PROGRAM ladder_logic_diagram 
VAR
	t2s: TIME := TIME#3S;
	t0s: TIME := TIME#0S;
	Timer: TON;
	input : BOOL;
	output : BOOL; 
	TON_Reset: TON;
	TON_set: TON;
	TON_0: TON;
	TON_Trig: TON;
	TON_Autonomous: TON;
	TON_Manual: TON;
	TON_Lock: TON;
	Robot_Mode_Timer: TON;
	liftUP: TON;
	liftDOWN: TON;
	load_button  AT %I* : BOOL ;
	load_active AT %Q*: BOOL;
	trigger AT %M* : BOOL ;
	T: TIME;
	TON_1: TON;
	TON2: TON;
	TON_3: TON;
	activate_time_read: BOOL;
	TON_4: TON;
	second_read_triggered: BOOL;
	first_read_triggered: BOOL;
	TON_5: TON;
	TON_6: TON;
	TON_7: TON;
END_VAR
VAR // added by the converter: edge detectors and wires of the graphical bodies
    _rt1 : R_TRIG;
    _w1 : BOOL;
END_VAR

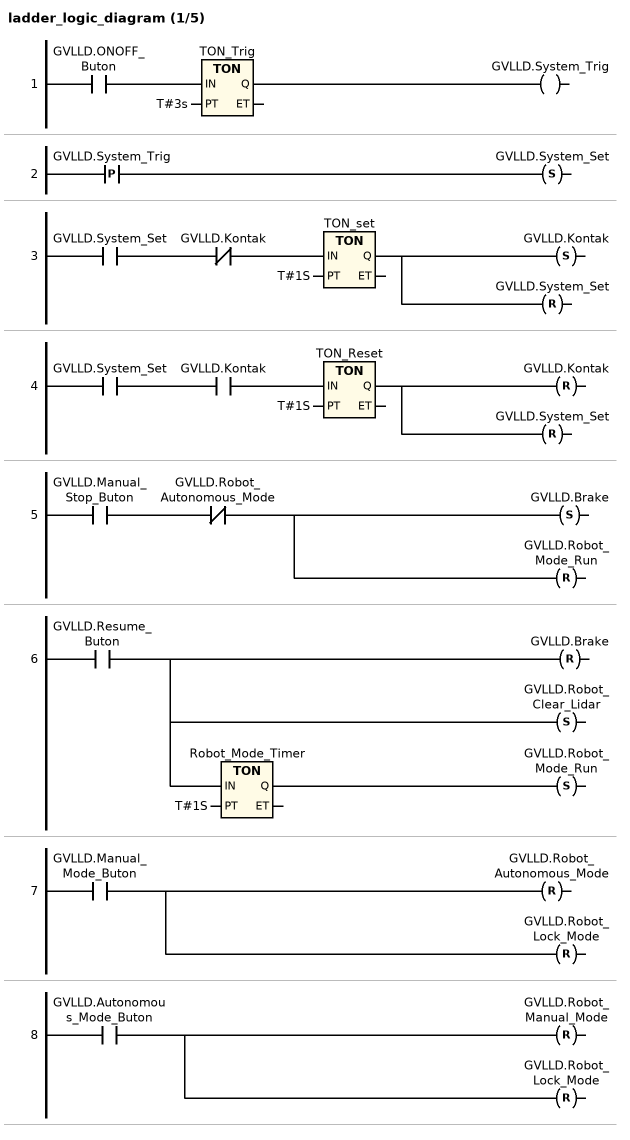
// NETWORK 1
TON_Trig(IN := GVLLD.ONOFF_Buton, PT := T#3s); // TON
GVLLD.System_Trig := TON_Trig.Q;

// NETWORK 2
_rt1(CLK := GVLLD.System_Trig);
GVLLD.System_Set S= _rt1.Q;

// NETWORK 3
TON_set(IN := GVLLD.System_Set AND NOT GVLLD.Kontak, PT := T#1S); // TON
GVLLD.Kontak S= TON_set.Q;
GVLLD.System_Set R= TON_set.Q;

// NETWORK 4
TON_Reset(IN := GVLLD.System_Set AND GVLLD.Kontak, PT := T#1S); // TON
GVLLD.Kontak R= TON_Reset.Q;
GVLLD.System_Set R= TON_Reset.Q;

// NETWORK 5
_w1 := GVLLD.Manual_Stop_Buton AND NOT GVLLD.Robot_Autonomous_Mode;
GVLLD.Brake S= _w1;
GVLLD.Robot_Mode_Run R= _w1;

// NETWORK 6
GVLLD.Brake R= GVLLD.Resume_Buton;
GVLLD.Robot_Clear_Lidar S= GVLLD.Resume_Buton;
Robot_Mode_Timer(IN := GVLLD.Resume_Buton, PT := T#1S); // TON
GVLLD.Robot_Mode_Run S= Robot_Mode_Timer.Q;

// NETWORK 7
GVLLD.Robot_Autonomous_Mode R= GVLLD.Manual_Mode_Buton;
GVLLD.Robot_Lock_Mode R= GVLLD.Manual_Mode_Buton;

// NETWORK 8
GVLLD.Robot_Manual_Mode R= GVLLD.Autonomous_Mode_Buton;
GVLLD.Robot_Lock_Mode R= GVLLD.Autonomous_Mode_Buton;

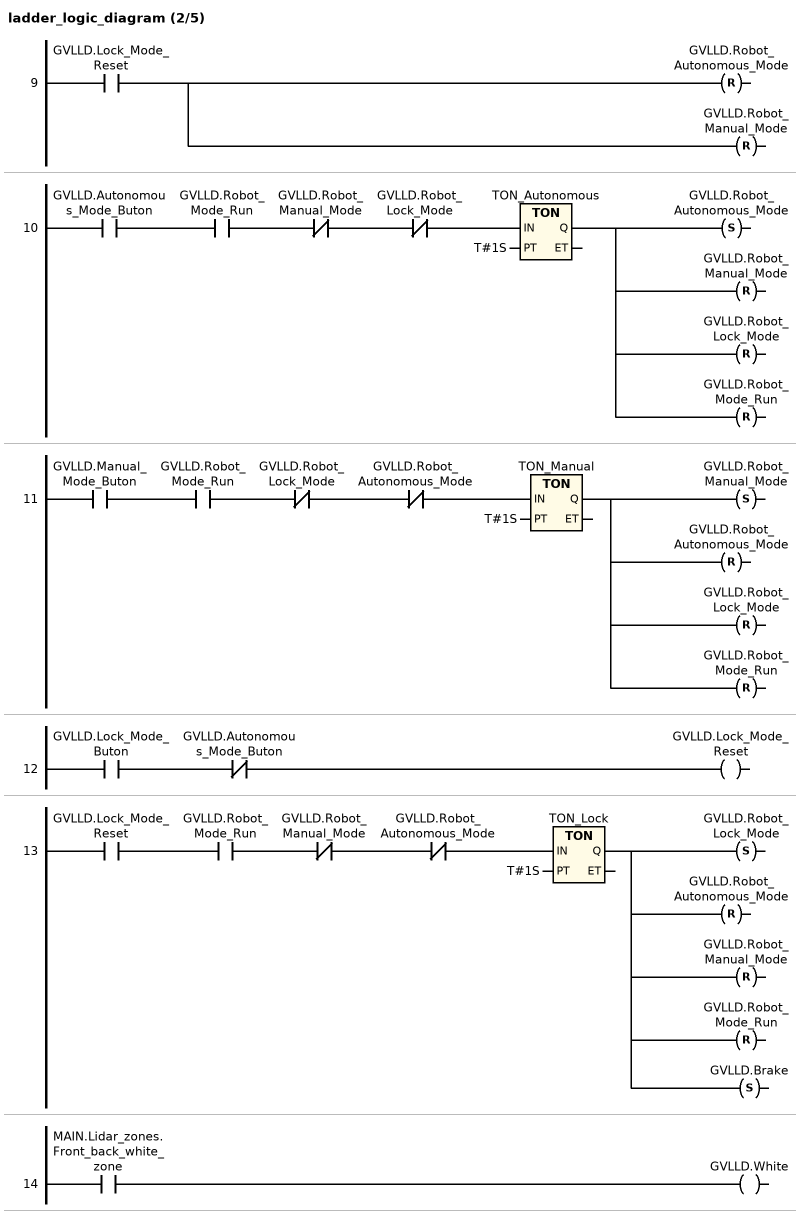
// NETWORK 9
GVLLD.Robot_Autonomous_Mode R= GVLLD.Lock_Mode_Reset;
GVLLD.Robot_Manual_Mode R= GVLLD.Lock_Mode_Reset;

// NETWORK 10
TON_Autonomous(IN := GVLLD.Autonomous_Mode_Buton AND GVLLD.Robot_Mode_Run AND NOT GVLLD.Robot_Manual_Mode AND NOT GVLLD.Robot_Lock_Mode, PT := T#1S); // TON
GVLLD.Robot_Autonomous_Mode S= TON_Autonomous.Q;
GVLLD.Robot_Manual_Mode R= TON_Autonomous.Q;
GVLLD.Robot_Lock_Mode R= TON_Autonomous.Q;
GVLLD.Robot_Mode_Run R= TON_Autonomous.Q;

// NETWORK 11
TON_Manual(IN := GVLLD.Manual_Mode_Buton AND GVLLD.Robot_Mode_Run AND NOT GVLLD.Robot_Lock_Mode AND NOT GVLLD.Robot_Autonomous_Mode, PT := T#1S); // TON
GVLLD.Robot_Manual_Mode S= TON_Manual.Q;
GVLLD.Robot_Autonomous_Mode R= TON_Manual.Q;
GVLLD.Robot_Lock_Mode R= TON_Manual.Q;
GVLLD.Robot_Mode_Run R= TON_Manual.Q;

// NETWORK 12
GVLLD.Lock_Mode_Reset := GVLLD.Lock_Mode_Buton AND NOT GVLLD.Autonomous_Mode_Buton;

// NETWORK 13
TON_Lock(IN := GVLLD.Lock_Mode_Reset AND GVLLD.Robot_Mode_Run AND NOT GVLLD.Robot_Manual_Mode AND NOT GVLLD.Robot_Autonomous_Mode, PT := T#1S); // TON
GVLLD.Robot_Lock_Mode S= TON_Lock.Q;
GVLLD.Robot_Autonomous_Mode R= TON_Lock.Q;
GVLLD.Robot_Manual_Mode R= TON_Lock.Q;
GVLLD.Robot_Mode_Run R= TON_Lock.Q;
GVLLD.Brake S= TON_Lock.Q;

// NETWORK 14
GVLLD.White := MAIN.Lidar_zones.Front_back_white_zone;

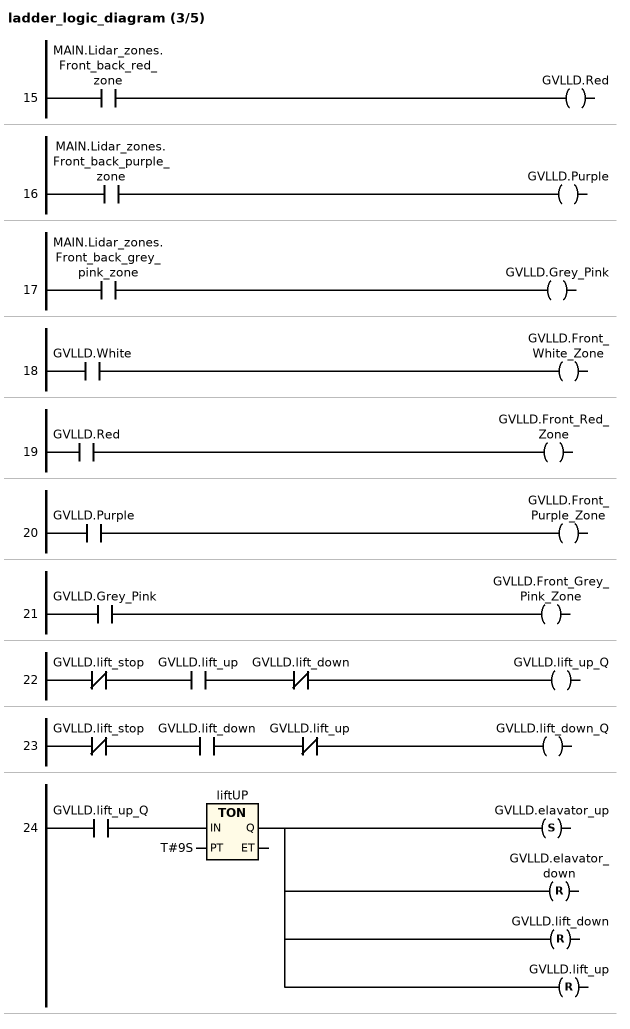
// NETWORK 15
GVLLD.Red := MAIN.Lidar_zones.Front_back_red_zone;

// NETWORK 16
GVLLD.Purple := MAIN.Lidar_zones.Front_back_purple_zone;

// NETWORK 17
GVLLD.Grey_Pink := MAIN.Lidar_zones.Front_back_grey_pink_zone;

// NETWORK 18
GVLLD.Front_White_Zone := GVLLD.White;

// NETWORK 19
GVLLD.Front_Red_Zone := GVLLD.Red;

// NETWORK 20
GVLLD.Front_Purple_Zone := GVLLD.Purple;

// NETWORK 21
GVLLD.Front_Grey_Pink_Zone := GVLLD.Grey_Pink;

// NETWORK 22
GVLLD.lift_up_Q := NOT GVLLD.lift_stop AND GVLLD.lift_up AND NOT GVLLD.lift_down;

// NETWORK 23
GVLLD.lift_down_Q := NOT GVLLD.lift_stop AND GVLLD.lift_down AND NOT GVLLD.lift_up;

// NETWORK 24
liftUP(IN := GVLLD.lift_up_Q, PT := T#9S); // TON
GVLLD.elavator_up S= liftUP.Q;
GVLLD.elavator_down R= liftUP.Q;
GVLLD.lift_down R= liftUP.Q;
GVLLD.lift_up R= liftUP.Q;

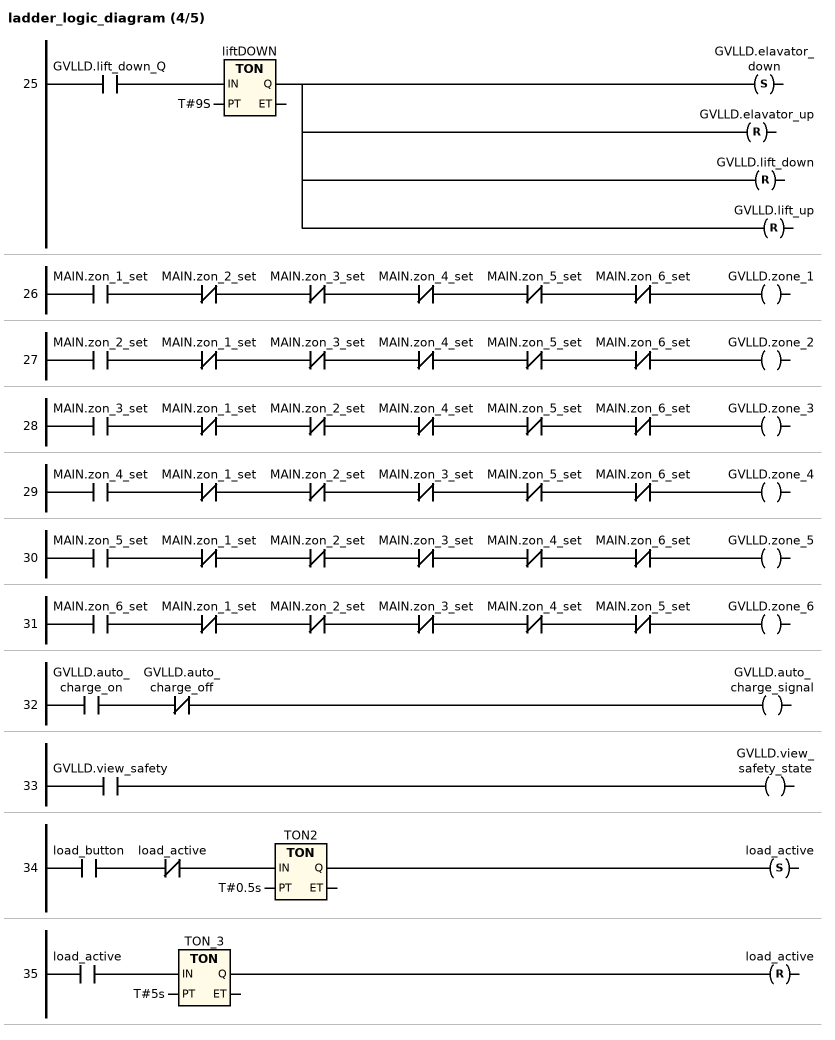
// NETWORK 25
liftDOWN(IN := GVLLD.lift_down_Q, PT := T#9S); // TON
GVLLD.elavator_down S= liftDOWN.Q;
GVLLD.elavator_up R= liftDOWN.Q;
GVLLD.lift_down R= liftDOWN.Q;
GVLLD.lift_up R= liftDOWN.Q;

// NETWORK 26
GVLLD.zone_1 := MAIN.zon_1_set AND NOT MAIN.zon_2_set AND NOT MAIN.zon_3_set AND NOT MAIN.zon_4_set AND NOT MAIN.zon_5_set AND NOT MAIN.zon_6_set;

// NETWORK 27
GVLLD.zone_2 := MAIN.zon_2_set AND NOT MAIN.zon_1_set AND NOT MAIN.zon_3_set AND NOT MAIN.zon_4_set AND NOT MAIN.zon_5_set AND NOT MAIN.zon_6_set;

// NETWORK 28
GVLLD.zone_3 := MAIN.zon_3_set AND NOT MAIN.zon_1_set AND NOT MAIN.zon_2_set AND NOT MAIN.zon_4_set AND NOT MAIN.zon_5_set AND NOT MAIN.zon_6_set;

// NETWORK 29
GVLLD.zone_4 := MAIN.zon_4_set AND NOT MAIN.zon_1_set AND NOT MAIN.zon_2_set AND NOT MAIN.zon_3_set AND NOT MAIN.zon_5_set AND NOT MAIN.zon_6_set;

// NETWORK 30
GVLLD.zone_5 := MAIN.zon_5_set AND NOT MAIN.zon_1_set AND NOT MAIN.zon_2_set AND NOT MAIN.zon_3_set AND NOT MAIN.zon_4_set AND NOT MAIN.zon_6_set;

// NETWORK 31
GVLLD.zone_6 := MAIN.zon_6_set AND NOT MAIN.zon_1_set AND NOT MAIN.zon_2_set AND NOT MAIN.zon_3_set AND NOT MAIN.zon_4_set AND NOT MAIN.zon_5_set;

// NETWORK 32
GVLLD.auto_charge_signal := GVLLD.auto_charge_on AND NOT GVLLD.auto_charge_off;

// NETWORK 33
GVLLD.view_safety_state := GVLLD.view_safety;

// NETWORK 34
TON2(IN := load_button AND NOT load_active, PT := T#0.5s); // TON
load_active S= TON2.Q;

// NETWORK 35
TON_3(IN := load_active, PT := T#5s); // TON
load_active R= TON_3.Q;

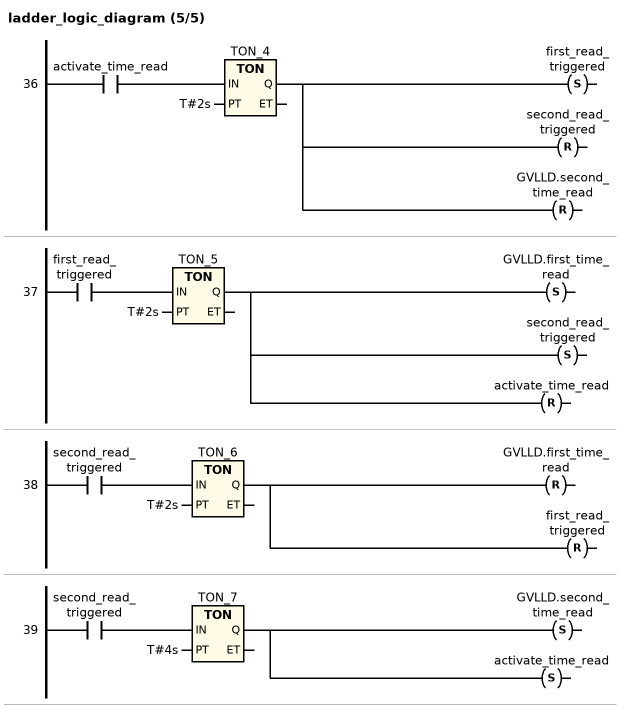
// NETWORK 36
TON_4(IN := activate_time_read, PT := T#2s); // TON
first_read_triggered S= TON_4.Q;
second_read_triggered R= TON_4.Q;
GVLLD.second_time_read R= TON_4.Q;

// NETWORK 37
TON_5(IN := first_read_triggered, PT := T#2s); // TON
GVLLD.first_time_read S= TON_5.Q;
second_read_triggered S= TON_5.Q;
activate_time_read R= TON_5.Q;

// NETWORK 38
TON_6(IN := second_read_triggered, PT := T#2s); // TON
GVLLD.first_time_read R= TON_6.Q;
first_read_triggered R= TON_6.Q;

// NETWORK 39
TON_7(IN := second_read_triggered, PT := T#4s); // TON
GVLLD.second_time_read S= TON_7.Q;
activate_time_read S= TON_7.Q;

END_PROGRAM

(* stored: Version 1.1.0.1, ProductVersion 3.1.4024.12
   POU ladder_logic_diagram: Id {8b49a9d5-a079-4a87-9de9-3f73f586a9cb}, SpecialFunc None *)
